// Mitsubishi GX Works2 project: IELET2103_PLSLab2   PLC: FX2N/FX2NC
// IELET2103_PLSLab2

// global labels: Global1
VAR_GLOBAL
  S0_Stopp : BOOL;
  S1_Start_Medurs : BOOL;
  S2_Start_Moturs : BOOL;
  Sekvens : WORD;
  F4_Motorvern : BOOL;
  H1_Driftsklar : BOOL;
  H2_Medurs : BOOL;
  H3_Moturs : BOOL;
  Medurs_K1 : BOOL;
  Moturs_K2 : BOOL;
  Startflagg_Medurs : BOOL;
  Feil_Aktiv : BOOL;
  Startflagg_Moturs : BOOL;
END_VAR

// task Task_01 (event TRUE, interval 0, priority 31): main, input, output

PROGRAM input
(* structured ladder/FBD written out as ST: instructions are called as NAME(EN, inputs, outputs); _pN, _eN, _tN stand for wires *)
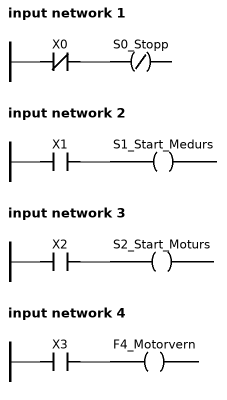
(* network 1 *)
S0_Stopp := NOT (NOT X0);
(* network 2 *)
S1_Start_Medurs := X1;
(* network 3 *)
S2_Start_Moturs := X2;
(* network 4 *)
F4_Motorvern := X3;
END_PROGRAM

PROGRAM main
VAR
  ton_1 : TON;
END_VAR
(* structured ladder/FBD written out as ST: instructions are called as NAME(EN, inputs, outputs); _pN, _eN, _tN stand for wires *)
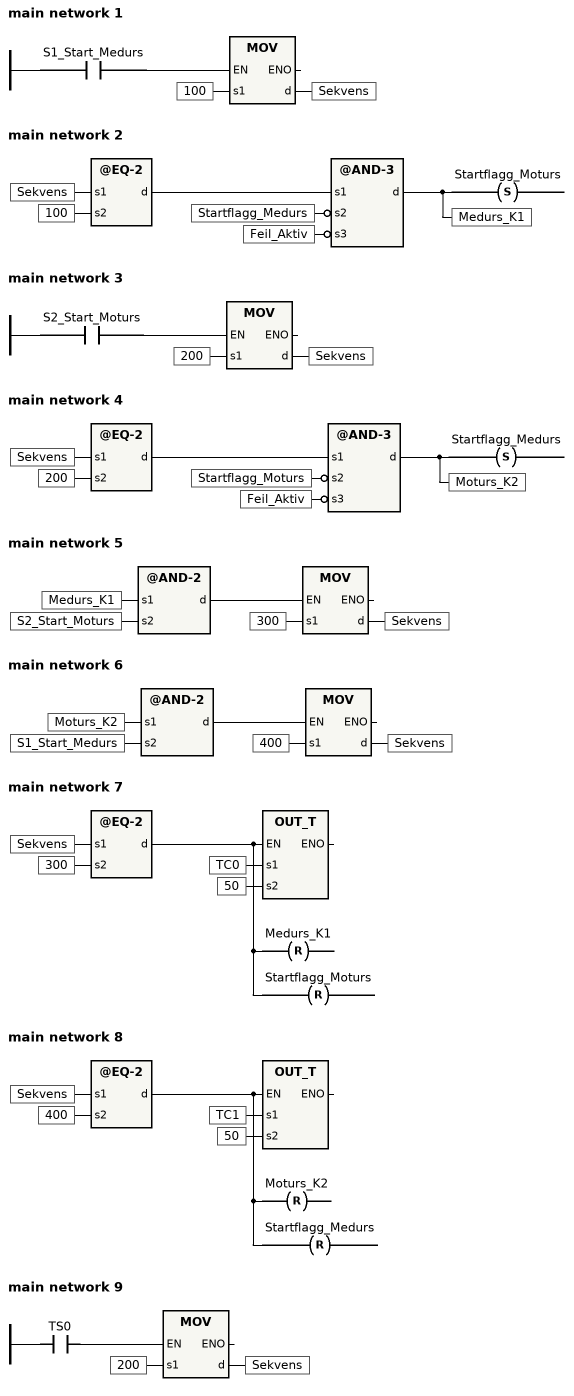
(* network 1 *)
MOV(S1_Start_Medurs, 100, Sekvens);
(* network 2 *)
_p1 := @AND-3(@EQ-2(Sekvens, 100), NOT Startflagg_Medurs, NOT Feil_Aktiv);
Medurs_K1 := _p1;
SET(_p1, Startflagg_Moturs);
(* network 3 *)
MOV(S2_Start_Moturs, 200, Sekvens);
(* network 4 *)
_p1 := @AND-3(@EQ-2(Sekvens, 200), NOT Startflagg_Moturs, NOT Feil_Aktiv);
Moturs_K2 := _p1;
SET(_p1, Startflagg_Medurs);
(* network 5 *)
MOV(@AND-2(Medurs_K1, S2_Start_Moturs), 300, Sekvens);
(* network 6 *)
MOV(@AND-2(Moturs_K2, S1_Start_Medurs), 400, Sekvens);
(* network 7 *)
_p1 := @EQ-2(Sekvens, 300);
OUT_T(_p1, TC0, 50);
RST(_p1, Medurs_K1);
RST(_p1, Startflagg_Moturs);
(* network 8 *)
_p1 := @EQ-2(Sekvens, 400);
OUT_T(_p1, TC1, 50);
RST(_p1, Moturs_K2);
RST(_p1, Startflagg_Medurs);
(* network 9 *)
MOV(TS0, 200, Sekvens);
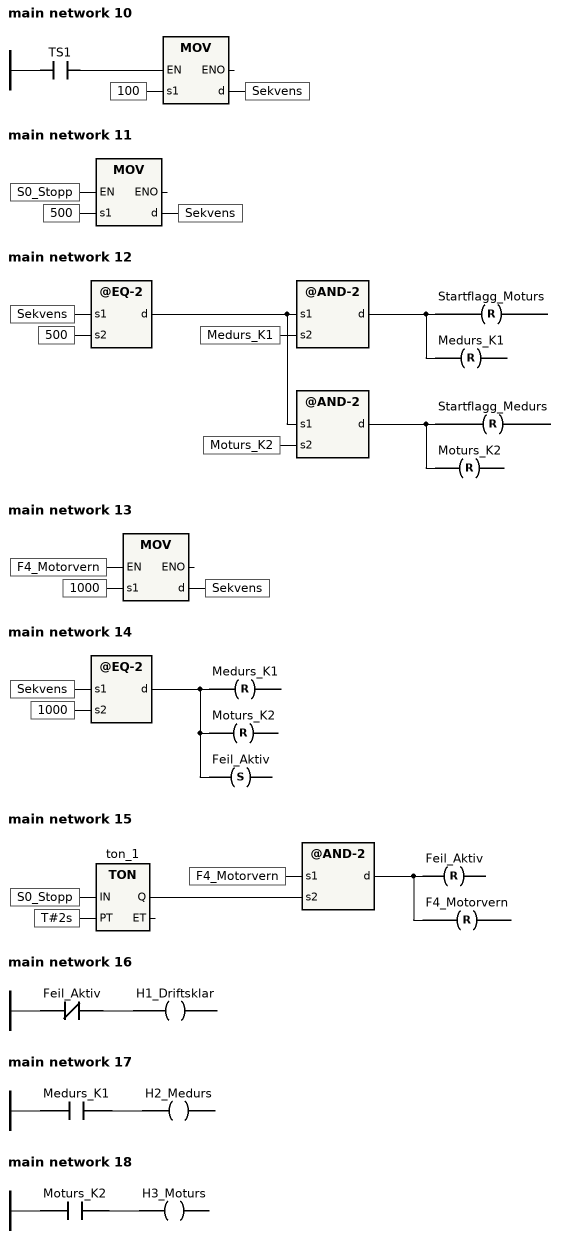
(* network 10 *)
MOV(TS1, 100, Sekvens);
(* network 11 *)
MOV(S0_Stopp, 500, Sekvens);
(* network 12 *)
_p1 := @EQ-2(Sekvens, 500);
_p2 := @AND-2(_p1, Medurs_K1);
RST(_p2, Startflagg_Moturs);
RST(_p2, Medurs_K1);
_p3 := @AND-2(_p1, Moturs_K2);
RST(_p3, Startflagg_Medurs);
RST(_p3, Moturs_K2);
(* network 13 *)
MOV(F4_Motorvern, 1000, Sekvens);
(* network 14 *)
_p1 := @EQ-2(Sekvens, 1000);
RST(_p1, Medurs_K1);
RST(_p1, Moturs_K2);
SET(_p1, Feil_Aktiv);
(* network 15 *)
ton_1(IN := S0_Stopp, PT := T#2s);
_p1 := @AND-2(F4_Motorvern, ton_1.Q);
RST(_p1, Feil_Aktiv);
RST(_p1, F4_Motorvern);
(* network 16 *)
H1_Driftsklar := NOT Feil_Aktiv;
(* network 17 *)
H2_Medurs := Medurs_K1;
(* network 18 *)
H3_Moturs := Moturs_K2;
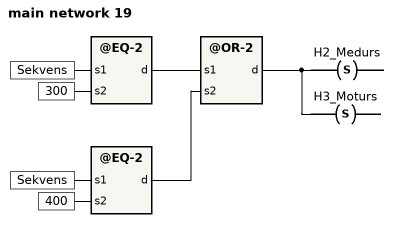
(* network 19 *)
_p1 := @OR-2(@EQ-2(Sekvens, 300), @EQ-2(Sekvens, 400));
SET(_p1, H2_Medurs);
SET(_p1, H3_Moturs);
END_PROGRAM

PROGRAM output
(* structured ladder/FBD written out as ST: instructions are called as NAME(EN, inputs, outputs); _pN, _eN, _tN stand for wires *)
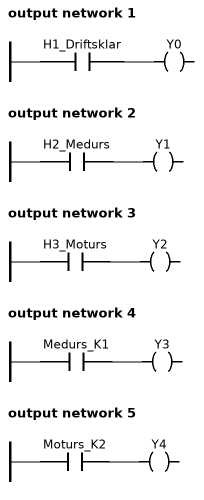
(* network 1 *)
Y0 := H1_Driftsklar;
(* network 2 *)
Y1 := H2_Medurs;
(* network 3 *)
Y2 := H3_Moturs;
(* network 4 *)
Y3 := Medurs_K1;
(* network 5 *)
Y4 := Moturs_K2;
END_PROGRAM
